PROGRAM P_Demo_FB_JsonSaxPrettyWriter
VAR
    fbFB_JsonSaxPrettyWriter : FB_JsonSaxPrettyWriter; // FB_JsonSaxPrettyWriter 实例
    initStatus : HRESULT; // FB 初始化状态
END_VAR

// =============================================================================
// 场景：调试 PLC ↔ 后端联调时把生成的 JSON 落盘成可读文件，方便 grep / diff。
// 价值：在 `FB_JsonSaxWriter` 基础上自动加缩进换行，调用代码完全相同。
// 验证：登录 PLC 在线写 bTrigger := TRUE 触发，monitor 返回值/输出参数。具体步骤见下方注释。
// 验证步骤：
//   1. 右键 PLC 项目下 POUs 文件夹 → Add → Existing Item → 选本 .TcPOU 文件
//   2. 引用 Tc3_JsonXml（References → Add library）
//   3. 编译 → 登录 → 运行；按 verify 注释里给出的在线写值操作
// =============================================================================

// 实例化 + 监视 initStatus，确认 FB 内部已初始化完成。
fbFB_JsonSaxPrettyWriter(
    initStatus => initStatus
);

// 进一步用法：参看 examples 目录下 FB_JsonSaxPrettyWriter_StartObject / FB_JsonSaxPrettyWriter_AddKeyString 等方法演示。

END_PROGRAM

(* stored: Version 1.1.0.1, ProductVersion 3.1.4024.5
   POU P_Demo_FB_JsonSaxPrettyWriter: Id {ebb82055-3dc7-5ecd-8ee9-5ed3e4a22b73}, SpecialFunc None *)
